Fanuc KAREL source: kt00297.KL

-- PROVISIONAL review KL for V940-1; original PC SHA256 287eaa7140659c917afb4b3453bc8790411e187d80601314ef8eb359b62b1ec3
-- Incomplete behavior may be omitted. Consult companion uncertainty JSON. Do not deploy.
PROGRAM KT00297
%NOLOCKGROUP
VAR
  R1 : REAL
  I2 : INTEGER
  OUT : BOOLEAN
BEGIN
  -- V9_ZERO_TABLE_METADATA_HINT layout=0001; no indexed target words; source/name/runtime held
  -- UNRESOLVED_PC offsets 5-16; opcodes 2E,23
  -- UNRESOLVED_PC offsets 21-32; opcodes 2E,23
  -- UNRESOLVED_PC offsets 37-57; opcodes 21,21,64,6E,23
  -- UNRESOLVED_PC offsets 62-66; opcodes 7F
END KT00297
